FUNCTION_BLOCK FB_Button
VAR_INPUT
	bprzyciskIn :BOOL;
	bAuto		:BOOL;
	
END_VAR
VAR_OUTPUT
	bprzyciskOut :BOOL;
END_VAR
VAR
	zbocze	:R_TRIG;
	thne: INT;
END_VAR


zbocze(CLK:=bprzyciskIn);
IF bAuto = TRUE THEN
	
bprzyciskOut:=FALSE;
	
END_IF

IF zbocze.Q=TRUE AND bprzyciskOut=TRUE  THEN 
	
bprzyciskOut:=FALSE;

ELSIF zbocze.Q=TRUE AND bprzyciskOut=FALSE  THEN


bprzyciskOut:=TRUE;

END_IF

END_FUNCTION_BLOCK

(* stored: Version 1.1.0.1, ProductVersion 3.1.4022.12
   POU FB_Button: Id {682f9806-5d7c-4ca4-ad4d-ca2d322c2bee}, SpecialFunc None *)
